{attribute 'linkalways'} 
{attribute 'no_explicit_call' := 'This FB is a CLASS and must be accessed using methods or properties'}
{attribute 'enable_dynamic_creation'}
FUNCTION_BLOCK EventHandlerItem IMPLEMENTS I_EventHandlerItem
VAR
	handler : I_EventHandler;
	_next : I_EventHandlerItem;
	_previous : I_EventHandlerItem;
END_VAR

METHOD PUBLIC Dispose
VAR_INPUT
END_VAR
__Delete(this);
END_METHOD

METHOD PUBLIC Emit
VAR_INPUT
	Event : I_Event;
END_VAR
IF handler = 0 THEN
	RETURN;
END_IF

handler.HandleEvent(Event);
END_METHOD

METHOD EqualTo : BOOL
VAR_INPUT
	Handler : I_EventHandler;
END_VAR
EqualTo := THIS^.handler = Handler;
END_METHOD

METHOD FB_init : BOOL
VAR_INPUT
	bInitRetains : BOOL; // if TRUE, the retain variables are initialized (warm start / cold start)
	bInCopyCode : BOOL;  // if TRUE, the instance afterwards gets moved into the copy code (online change)
	Handler : I_EventHandler;
END_VAR
THIS^.handler := Handler;
END_METHOD

PROPERTY PUBLIC Next : I_EventHandlerItem
GET
Next := _next;
END_GET
SET
_next := Next;
END_SET
END_PROPERTY

PROPERTY PUBLIC Previous : I_EventHandlerItem
GET
Previous := _previous;
END_GET
SET
_previous := Previous;
END_SET
END_PROPERTY

END_FUNCTION_BLOCK

(* stored: Version 1.1.0.1, ProductVersion 3.1.4024.12
   POU EventHandlerItem: Id {2aa43558-6b83-4717-b221-d389f1b91280}, SpecialFunc None
   Folder Constructor: Id {f9475fe6-abfb-417a-9bac-6dc8e072a5b7}
   Method Dispose: Id {903a4fcb-c448-4581-897d-aff7b80d98d1}
   Method Emit: Id {a08bbc57-5907-4ad0-a169-808f181d1d31}
   Method EqualTo: Id {ff72ec5b-86e4-4328-9b69-db9c34224bd1}
   Method FB_init: Id {88b9db40-2c85-4ec5-8e0c-4eb1a00785ff}
   Property Next: Id {4c23dc9f-2d75-4984-88a6-1733b8118057}
   Get Get: Id {4aabe7ba-0f2b-4a3e-8c52-9bc5d1af8e98}
   Set Set: Id {1b9c21b5-7235-458c-8bff-ea3142f4bc7e}
   Property Previous: Id {ae1cf066-cd4f-41d2-ab8e-d4ae0e4ffd34}
   Get Get: Id {93ec4aaa-a36e-404c-880a-443bdd19e823}
   Set Set: Id {15c32a9c-3046-494f-a5ce-7da79a20b13f} *)
